// TIA Portal project "2022.05.16_用户界面" (V17)

(* hardware
DEVICE "S7-1500/ET200MP station_1"  S7-1500 station
   slot 0: "导轨_0"  Rack  6ES7 590-1***0-0AA0
   slot 1: "PLC_1500"  CPU 1516-3 PN/DP  6ES7 516-3AN00-0AB0  V1.7
      slot 3: "CPU 显示_1"  6ES7591-1BA00-0AA0
      slot 32768: "PROFINET 接口_1"  X1
         slot 32769: "端口_1"  X1 P1
         slot 32770: "端口_2"  X1 P2
      slot 33024: "PROFINET 接口_2"  X2
         slot 33025: "端口_1"  X2 P1
      slot 33280: "DP 接口_1"  X3
DEVICE "HMI_1"  TP1200 Comfort
   slot 0: "HMI_1"  TP1200 Comfort  6AV2 124-0MC01-0AX0  17.0.0.0
   slot 1: "HMI_RT_1"  TP1200 Comfort  6AV2 124-0MC01-0AX0  17.0.0.0
   slot 5: "HMI_1.IE_CP_1"  PROFINET Interface  17.0.0.0
      slot 1: "PROFINET Interface_1"  PROFINET Interface
         slot 1: "Port_1"  Port
         slot 2: "Port_2"  Port
   slot 7: "HMI_1.MPI/DP_CP_1"  MPI/DP Interface  17.0.0.0
*)

// ===== PLC "PLC_1500"  CPU 1516-3 PN/DP =====

ORGANIZATION_BLOCK "Main"   // OB1, LAD, ProgramCycle
TITLE = "Main Program Sweep (Cycle)"
{ S7_Optimized_Access := 'TRUE' }
VERSION : 0.1
   VAR_INPUT
      Initial_Call : Bool;   // Initial call of this OB
      Remanence : Bool;   // =True, if remanent data are available
   END_VAR
BEGIN
END_ORGANIZATION_BLOCK

(* ===== HMI "HMI_RT_1" =====
system functions are stored by id; their names below are inferred from use
connection "PLC_1500": ETHERNET, S7_1500_OMS
connection "Connection_1": ETHERNET, S7_1500_OMS

HMI tags "默认变量表"
   "Tag_ScreenNumber" : UInt, internal

HMI tags "变量表_1"
   "按钮1控制" : Bool, internal
   "按钮2控制" : Bool, internal
   "按钮3控制" : Bool, internal

screen "根画面" 1280x740, template "模板_1"
   on GenerateScreen: SetTag("Tag_ScreenNumber", 1)
   TextField "文本域_1" at 244,85 size 203x25; Text '用户管理的层级关系'
   TextField "文本域_2" at 275,162 size 149x21; Text '权限（可以多个）'
   TextField "文本域_3" at 282,263 size 131x21; Text '组（可以多个）'
   TextField "文本域_4" at 374,212 size 239x21; Text '一个用户组可以拥有多种权限'
   TextField "文本域_5" at 275,370 size 149x21; Text '用户（可以多个）'
   TextField "文本域_6" at 373,319 size 239x21; Text '一个用户组可以拥有多个用户'
   TextField "文本域_7" at 257,460 size 383x21; Text '注：单个用户必须拥有自己的密码、注销时间等'
   UserView "用户视图_1" at 637,98 size 614x392
   Button "按钮_1" at 720,50 size 77x32; TextOff '按钮1'; Authorization "User administration"
      Appearance <- "按钮1控制"
      on Click: InvertBit("按钮1控制")
   Button "按钮_2" at 856,52 size 77x32; TextOff '按钮2'; Authorization "Monitor"
      on Click: InvertBit("按钮2控制")
      Appearance <- "按钮2控制"
   Button "按钮_3" at 987,53 size 77x32; TextOff '按钮3'; Authorization "Operate"
      Appearance <- "按钮3控制"
      on Click: InvertBit("按钮3控制")
   TextField "文本域_8" at 737,22 size 59x21; Text '管理员'
   TextField "文本域_9" at 871,23 size 41x21; Text '监视'
   TextField "文本域_10" at 1003,23 size 41x21; Text '操作'

Template "模板_1" 1280x740
   Button "退出" at 1200,679 size 78x59; TextOff '退出'; PictureOff "ExitRuntime_TP1200_Comfort_TR"; PictureOn "ExitRuntime_TP1200_Comfort_TR"
      on Release: StopRuntime(0)
   Button "Template_Button" at 1120,679 size 78x59; TextOff 'Text'
   Button "Template_Button_1" at 1040,679 size 78x59; TextOff 'Text'
   Button "Template_Button_2" at 960,679 size 78x59; TextOff 'Text'
   Button "Template_Button_3" at 880,679 size 78x59; TextOff 'Text'
   Button "Template_Button_4" at 800,679 size 78x59; TextOff 'Text'
   Button "Template_Button_5" at 720,679 size 78x59; TextOff 'Text'
   Button "Template_Button_6" at 640,679 size 78x59; TextOff 'Text'
   Button "Template_Button_7" at 561,679 size 78x59; TextOff 'Text'
   Button "Template_Button_8" at 481,679 size 78x59; TextOff 'Text'
   Button "Template_Button_9" at 401,679 size 78x59; TextOff 'Text'
   Button "Template_Button_10" at 321,679 size 78x59; TextOff 'Text'
   Button "Template_Button_11" at 241,679 size 78x59; TextOff 'Text'
   Button "Template_Button_12" at 161,679 size 78x59; TextOff 'Text'
   Button "Template_Button_13" at 81,679 size 78x59; TextOff 'Text'
   Button "起始画面" at 1,679 size 78x59; TextOff '起始画面'; PictureOff "NavigateHome_TP1200_Comfort_TR"; PictureOn "NavigateHome_TP1200_Comfort_TR"
      on Release: ActivateScreen("根画面", 0)
*)